TYPE Gauge_Type: ( PG722B := 0, IG903 := 1 , PG907 := 2 , IG909:= 3 ,PG925 := 4 );
(* This enumeration should match up with the EDM MUX button on the vacuum gauge expert controls screen *)
END_TYPE

(* stored: Version 1.1.0.1, ProductVersion 3.1.0.24
   DUT Gauge_Type: Id {c777043f-0b38-4846-b2d2-725c1a5388f6} *)
